// TIA Portal V20 export
DATA_BLOCK "EVTLOG"   // DB950
{ S7_Optimized_Access := 'FALSE' }
VERSION : 0.1
// Standard access : gr-console reads by S7 (DB950), layout checked by LayoutSig. Writer : "EvtWrite" only
// stored: AutoNumber false, DBAccessibleFromOPCUA true, DBAccessibleFromWebserver true, IsOnlyStoredInLoadMemory false, IsWriteProtectedInAS false
   VAR
      LayoutSig : DWord := 16#7915_BD0A;   // gr-contract gen-sig, do not edit
      Total : UDInt;   // rows written since boot = Seq of the newest row
      Head : Int;   // next write index (newest = Entry[Head-1])
      BootId : UInt;   // EVTWATCH.BootCount (low 16 bit), new epoch on change
      Dropped : UDInt;   // rows refused by Cfg.MaxPerScan
      Stat : Struct
         RunUs : UDInt;   // UL_EvtPre + UL_EvtWatch, last scan (µs)
         MaxRunUs : UDInt;   // console may reset
         MaxPerScanHit : UDInt;   // scans that reached Cfg.MaxPerScan
      END_STRUCT;
      Cfg : Struct   // console writable
         MinLevel : USInt := 2;   // EVT_LVL_* : lower levels are not written
         CatMask : DWord := 16#0003_FFFE;   // bit n = EVT_CAT id n
         MaxPerScan : Int := 32;
      END_STRUCT;
      Now : Struct   // per-scan context (UL_EvtPre)
         "Time" : DTL;
         Ctx : UDInt;
         Count : Int;
      END_STRUCT;
      Entry { S7_SetPoint := 'True'} : Array[0.."EVT_LAST"] of "EVT_Entry";
   END_VAR
BEGIN
END_DATA_BLOCK
